// TIA Portal V19 export
FUNCTION_BLOCK "TYPIC_C302_IF_LKM"   // FB103, FBD
TITLE = TYPIC_C302_IF_LKM: Luchtkwaliteitsmeter
{ S7_Optimized_Access := 'TRUE' }
AUTHOR : OCOTECH
FAMILY : Typical
NAME : C302.701
// Logisch Object Besturing: C302.701
// 
// De interne functie luchtkwaliteitsmeting verzorgt de interne besturing en bewaking van een luchtkwaliteitsmeter.
// stored: MemoryReserve 10, SetENOAutomatically false
   VAR_INPUT
      EXT_AUT { ExternalAccessible := 'False'; ExternalVisible := 'False'; ExternalWritable := 'False'} : Bool;   // Externe (hoofd) beveiliging (1 = OK)
      EXT_HW { ExternalAccessible := 'False'; ExternalVisible := 'False'; ExternalWritable := 'False'} : Bool;   // Sturings hardware (PLC) bewaking (1 = OK)
      IN_AUT_C302 { ExternalAccessible := 'False'; ExternalVisible := 'False'; ExternalWritable := 'False'} : Bool;   // Beveiligingen: serie geschakelde terugmelding (1 = OK)
      IN_STS { ExternalAccessible := 'False'; ExternalVisible := 'False'; ExternalWritable := 'False'} : Bool;   // TRUE = Aan / FALSE = Uit
      IN_STO { ExternalAccessible := 'False'; ExternalVisible := 'False'; ExternalWritable := 'False'} : Bool;   // TRUE = OK / FALSE = Storing
      IN_MWA { ExternalAccessible := 'False'; ExternalVisible := 'False'; ExternalWritable := 'False'} : Word;   // Meetwaarde [m-1]
      CFG_MAX_SWA { ExternalAccessible := 'False'; ExternalVisible := 'False'; ExternalWritable := 'False'} : Real;   // Waarde doe toegekend wordt aan LKM_MWA als maximumwaarde voor de meeteenheid [m-1]
      CFG_MIN_SWA { ExternalAccessible := 'False'; ExternalVisible := 'False'; ExternalWritable := 'False'} : Real;   // Waarde doe toegekend wordt aan LKM_MWA als minimumwaarde voor de meeteenheid [m-1]
   END_VAR
   VAR_OUTPUT
      VAR_IF_LKM { ExternalAccessible := 'False'; ExternalVisible := 'False'; ExternalWritable := 'False'} : "C302_VAR_IF_LKM_TYPIC";   // Struct met alle variabelen naar bovenliggende functies
   END_VAR
   VAR
      STO { ExternalWritable := 'False'} : Struct   // Storingen
         A001 : Bool;   // Luchtkwaliteitsmeter niet aangeschakeld
         A002 : Bool;   // Draadbreuk analoge meting
         A003 : Bool;   // Meetbereik overschreden
         A004 : Bool;   // Luchtkwaliteitsmeter geeft storing
      END_STRUCT;
      VAR { ExternalWritable := 'False'} : Struct   // Variabelen
         LKM_MWA { ExternalAccessible := 'False'; ExternalVisible := 'False'} : Real;   // Meetwaarde [m-1]
         EXT_AUT { ExternalAccessible := 'False'; ExternalVisible := 'False'} : Bool;   // Externe (hoofd) beveiliging aangesproken
         EXT_HW { ExternalAccessible := 'False'; ExternalVisible := 'False'} : Bool;   // Sturings hardware (PLC) in storing
      END_STRUCT;
   END_VAR
BEGIN

REGION Network 1: START
END_REGION

REGION Network 2: +++ Verwerking analoge meting +++
   // Verwerking analoge meting naar een meetwaarde (k-waarde) en detectie storingen van de luchtkwaliteitsmeter.
END_REGION

REGION Network 3 (SCL): EINDE
   // Variabelen van intern scada rakvlak naar outputs copieren
   #VAR_IF_LKM.LKM_MWA := #VAR.LKM_MWA;
   #VAR_IF_LKM.EXT_AUT := #VAR.EXT_AUT;
   #VAR_IF_LKM.EXT_HW := #VAR.EXT_HW;
   #VAR_IF_LKM.STO := #STO;
END_REGION
END_FUNCTION_BLOCK
